Universal Robots URScript: Define_Waypoints_Block.script

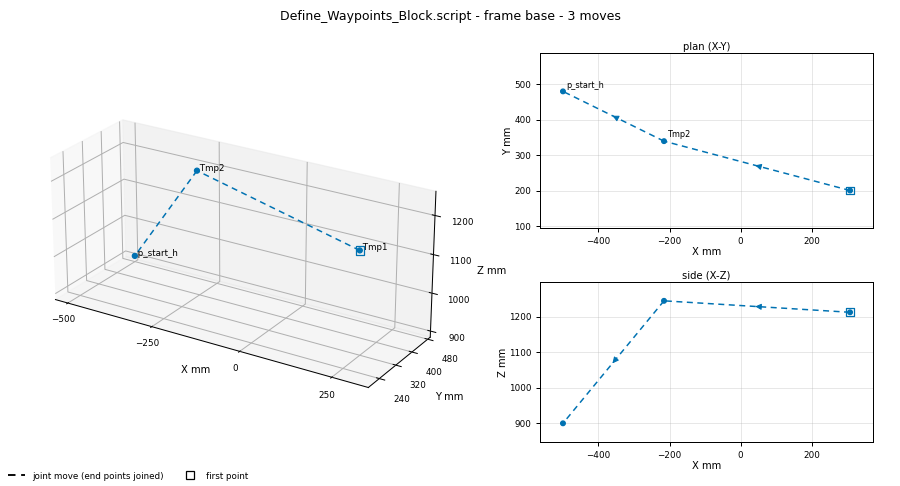
[picture p0: tool path of Define_Waypoints_Block.script in frame base, 3 of 4 moves have a stored position in this frame; points joined in program order, loops and branches not executed]
def Define_Waypoints_Block():
  global _hidden_verificationVariable=0
  step_count_e07f7cfb_3ea7_495d_acb1_b26853f0fbb6 = 0.0
  thread Step_Counter_Thread_c9ae2efd_e4bf_471e_9d91_553d842f2b7f():
    while (True):
      step_count_e07f7cfb_3ea7_495d_acb1_b26853f0fbb6 = step_count_e07f7cfb_3ea7_495d_acb1_b26853f0fbb6 + 1.0
      sync()
    end
  end
  run Step_Counter_Thread_c9ae2efd_e4bf_471e_9d91_553d842f2b7f()
  motion_version_set(2)
  set_tcp(p[0.0,0.0,0.0,0.0,0.0,0.0])
  tool_wrench_limit_disable()
  set_safety_mode_transition_hardness(1)
  set_gravity([0.0, -9.82, 6.013015783813504E-16])
  set_standard_analog_input_domain(0, 1)
  set_standard_analog_input_domain(1, 1)
  set_tool_analog_input_domain(0, 1)
  set_tool_analog_input_domain(1, 1)
  set_analog_outputdomain(0, 0)
  set_analog_outputdomain(1, 0)
  set_input_actions_to_default()
  set_target_payload(1.970000, [-0.003000, -0.010000, 0.017000], [0.004766, 0.004766, 0.004766, 0.000000, 0.000000, 0.000000])
  set_tool_communication(False, 115200, 0, 1, 1.5, 3.5)
  set_tool_output_mode(0)
  set_tool_digital_output_mode(0, 2)
  set_tool_digital_output_mode(1, 2)
  set_tool_voltage(0)
  global line_length=0
  global line_incr=0
  global avoid_start=0
  global avoid_end=0
  global avoid_gap=0
  global Plane_1=p[0.0,0.58,0.0,-1.5707963267948963,-2.9874637964168546E-16,-2.9874637964168546E-16]
  # begin: URCap Installation Node
  #   Source: UR Connect, 2.3.8, Universal Robots
  #   Type: UR Connect
  myurRPC = rpc_factory("xmlrpc","http://127.0.0.1:40474")
  # end: URCap Installation Node
  global Tmp1_p=p[.308197528239, .200952848898, 1.212577409890, -1.500617001311, .096591502570, -1.942084517693]
  global Tmp1_q=[2.9922775051327015, -1.8204617628859179, 0.7854625361952244, 0.6468829346793701, 1.081932385811806, 2.2461432469487175]
  global Tmp2_p=p[-.215537331320, .339862281058, 1.244844388379, -1.453965512348, -.560096017943, -.789013712763]
  global Tmp2_q=[3.0693981647491455, -2.002010484735006, 0.261266056691305, 0.8101395803638916, 0.07373906672000885, 3.208488702774048]
  global p_start_h_p=p[-.500000000000, .480000000000, .900000000000, .000041430133, 2.221422900018, 2.221426094739]
  global p_start_h_q=[2.863824951205764, -1.673476762916664, -1.6620415782888411, 0.18480899190657585, 0.2846715173802181, 3.150983641616914]
  $ 2 "Robot Program"
  $ 3 "Home"
  movej([1.5704206228256226, -1.3090128761580964, 2.443455998097555, -1.134462670688965, 1.5708153247833252, 1.5707963267948966], a=1.3962634015954636, v=1.0471975511965976)
  $ 4 "MoveJ"
  $ 5 "Tmp1" "breakAfter"
  movej(get_inverse_kin(Tmp1_p, qnear=Tmp1_q), a=1.3962634015954636, v=1.0471975511965976)
  $ 6 "Tmp2" "breakAfter"
  movej(get_inverse_kin(Tmp2_p, qnear=Tmp2_q), a=1.3962634015954636, v=1.0471975511965976)
  $ 7 "MoveJ"
  $ 8 "p_start_h" "breakAfter"
  movej(get_inverse_kin(p_start_h_p, qnear=p_start_h_q), a=1.3962634015954636, v=1.0471975511965976)
  $ 9 "Script: apply_force_logic.script"
  # This is the Script-node source for Benoit/apply_force.urp.
  # Keep the source name different from apply_force.script because PolyScope
  # generates apply_force.script automatically when it saves apply_force.urp.

  # ---------- Configuration ----------
  register = 42

  # Global variables appear with live values in PolyScope's Variables pane.
  global apply_force_phase = "Setting program variables"
  global apply_force_max_distance = read_input_float_register(43)
  global apply_force_contact_threshold = read_input_float_register(44)
  global apply_force_holding_force = read_input_float_register(45)
  global apply_force_simulation = read_input_integer_register(46) == 1
  global apply_force_force_reached = False

  # Fixed safety settings, identical to move50mm_force.script.
  max_approach_speed = 0.020
  contact_timeout = 10.0

  return_speed = 0.020
  return_acceleration = 0.100

  # Status:
  # 0 = initialized / completed
  # 1 = force reached (real or simulated); waiting for Python acknowledgement
  # 2 = maximum distance reached without contact
  # 3 = acknowledgement timeout

  write_output_integer_register(register, 0)

  # Reject acknowledgement remaining from an earlier run
  while read_input_integer_register(register) != 0:
      sync()
  end

  start_pose = get_actual_tcp_pose()
  force_frame = start_pose

  zero_ftsensor()
  sleep(0.2)

  contact_detected = False
  maximum_reached = False

  # Approach along the starting TCP Z+ direction
  apply_force_phase = "Moving to reach contact force"

  while (contact_detected == False) and (maximum_reached == False):

      force_mode(
          force_frame,
          [0, 0, 1, 0, 0, 0],
          [0, 0, apply_force_holding_force, 0, 0, 0],
          2,
          [0.010, 0.010, max_approach_speed, 0.10, 0.10, 0.10]
      )

      current_pose = get_actual_tcp_pose()
      relative_pose = pose_trans(pose_inv(start_pose), current_pose)
      travelled_z = relative_pose[2]

      measured_force = force()

      if measured_force >= apply_force_contact_threshold:
          contact_detected = True
      elif travelled_z >= apply_force_max_distance:
          maximum_reached = True
      end

      sync()
  end

  # In simulation, reaching maximum distance is reported as force reached. Stop
  # force mode first so the robot cannot move beyond the configured distance while
  # Python performs the simulated hold/acknowledgement sequence.
  force_mode_stopped = False

  if contact_detected:
      apply_force_force_reached = True
  elif maximum_reached and apply_force_simulation:
      apply_force_force_reached = True
      end_force_mode()
      stopl(1.0)
      sleep(0.1)
      force_mode_stopped = True
  end

  if apply_force_force_reached:

      if contact_detected:
          apply_force_phase = "Force reached"
      else:
          apply_force_phase = "Maximum displacement reached; simulating force reached"
      end
      write_output_integer_register(register, 1)

      acknowledged = False
      timed_out = False
      elapsed_time = 0.0

      # Maintain real force while waiting for Python. In simulation, force mode was
      # already stopped at maximum distance and this loop only waits for the same
      # acknowledgement, allowing the rest of the workflow to be tested.
      if contact_detected:
          apply_force_phase = "Waiting for end of force hold"
      else:
          apply_force_phase = "Waiting for end of simulated hold"
      end

      while (acknowledged == False) and (timed_out == False):

          if contact_detected:
              force_mode(
                  force_frame,
                  [0, 0, 1, 0, 0, 0],
                  [0, 0, apply_force_holding_force, 0, 0, 0],
                  2,
                  [0.010, 0.010, max_approach_speed, 0.10, 0.10, 0.10]
              )
          end

          if read_input_integer_register(register) == 1:
              acknowledged = True
          end

          elapsed_time = elapsed_time + get_steptime()

          if elapsed_time >= contact_timeout:
              timed_out = True
          end

          sync()
      end

      if timed_out:
          apply_force_phase = "Force hold acknowledgement timed out"
          write_output_integer_register(register, 3)
      else:
          apply_force_phase = "Force hold completed"
      end

  else:

      apply_force_phase = "Maximum displacement reached"
      write_output_integer_register(register, 2)

  end

  if force_mode_stopped == False:
      end_force_mode()
      stopl(1.0)
      sleep(0.1)
  end

  apply_force_phase = "Moving back to initial position"

  movel(
      start_pose,
      a=return_acceleration,
      v=return_speed
  )

  apply_force_phase = "Initial position reached"

  write_output_integer_register(register, 0)

  apply_force_phase = "Cycle completed"
end
